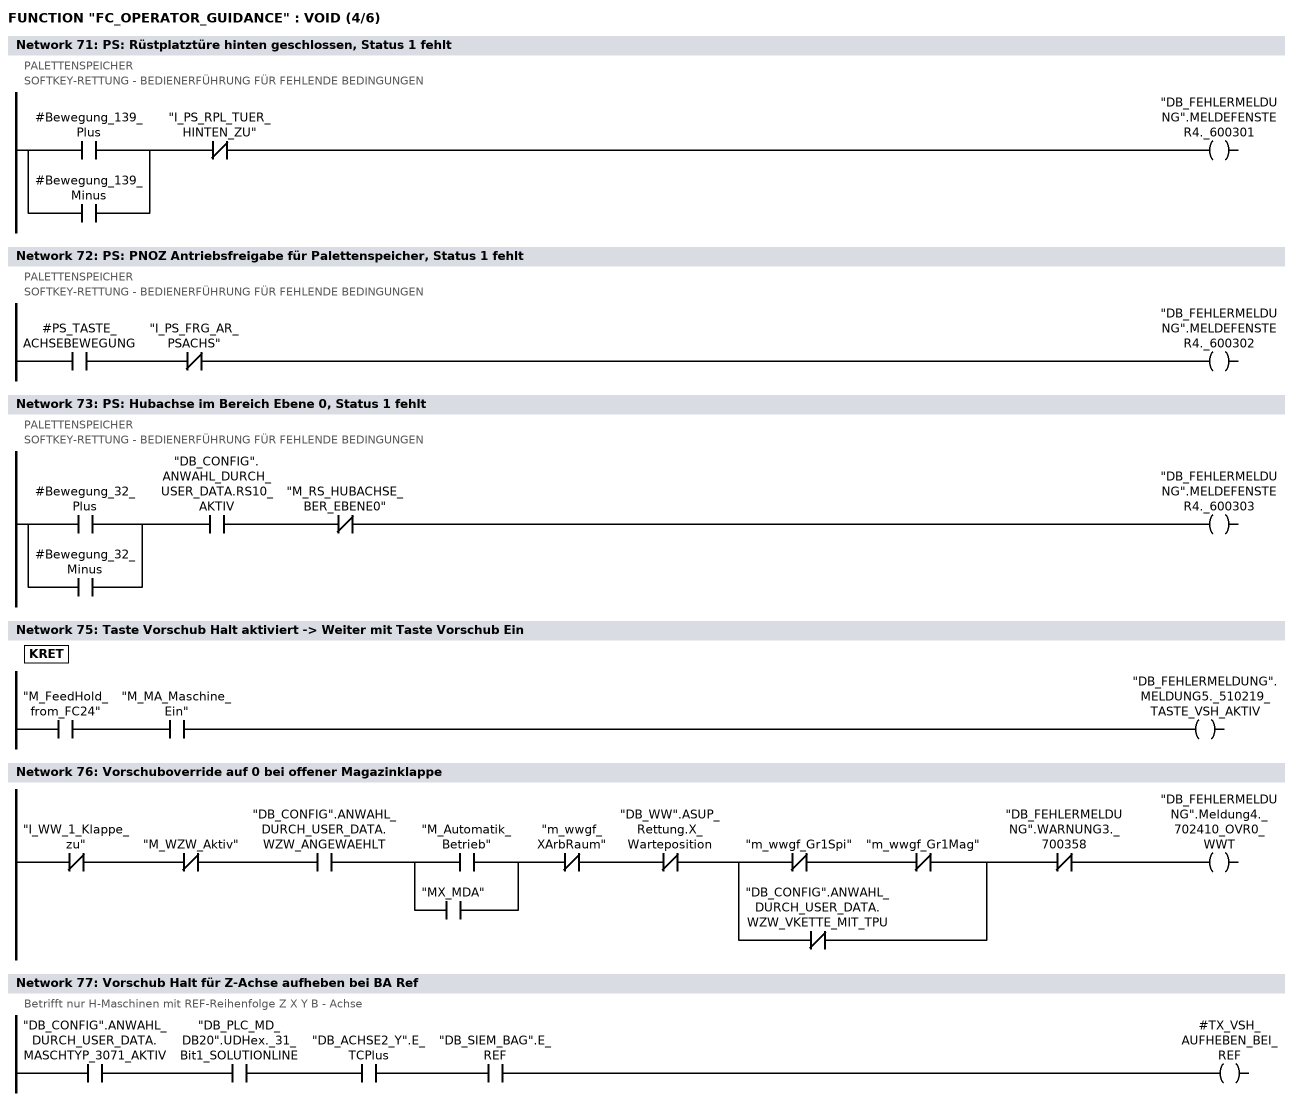
      U(    ;
      O     #Bewegung_139_Plus;
      O     #Bewegung_139_Minus;
      )     ;
      UN    "I_PS_RPL_TUER_HINTEN_ZU";
      =     "DB_FEHLERMELDUNG".MELDEFENSTER4._600301;
NETWORK
TITLE =PS: PNOZ Antriebsfreigabe für Palettenspeicher, Status 1 fehlt
//PALETTENSPEICHER
//SOFTKEY-RETTUNG - BEDIENERFÜHRUNG FÜR FEHLENDE BEDINGUNGEN
      U     #PS_TASTE_ACHSEBEWEGUNG;
      UN    "I_PS_FRG_AR_PSACHS";
      =     "DB_FEHLERMELDUNG".MELDEFENSTER4._600302;
NETWORK
TITLE =PS: Hubachse im Bereich Ebene 0, Status 1 fehlt
//PALETTENSPEICHER
//SOFTKEY-RETTUNG - BEDIENERFÜHRUNG FÜR FEHLENDE BEDINGUNGEN
      U(    ;
      O     #Bewegung_32_Plus;
      O     #Bewegung_32_Minus;
      )     ;
      U     "DB_CONFIG".ANWAHL_DURCH_USER_DATA.RS10_AKTIV;
      UN    "M_RS_HUBACHSE_BER_EBENE0";
      =     "DB_FEHLERMELDUNG".MELDEFENSTER4._600303;
NETWORK
TITLE =VORSCHUBSPERREN / VORSCHUB HALT

NETWORK
TITLE =Taste Vorschub Halt aktiviert -> Weiter mit Taste Vorschub Ein

KRET: U     "M_FeedHold_from_FC24";
      U     "M_MA_Maschine_Ein";
      =     "DB_FEHLERMELDUNG".MELDUNG5._510219_TASTE_VSH_AKTIV;
NETWORK
TITLE =Vorschuboverride auf 0 bei offener Magazinklappe

      UN    "I_WW_1_Klappe_zu";
      UN    "M_WZW_Aktiv";
      U     "DB_CONFIG".ANWAHL_DURCH_USER_DATA.WZW_ANGEWAEHLT;
      U(    ;
      O     "M_Automatik_Betrieb";
      O     "MX_MDA";
      )     ;
      UN    "m_wwgf_XArbRaum";
      UN    "DB_WW".ASUP_Rettung.X_Warteposition;
      U(    ;
      UN    "m_wwgf_Gr1Spi";
      UN    "m_wwgf_Gr1Mag";
      ON    "DB_CONFIG".ANWAHL_DURCH_USER_DATA.WZW_VKETTE_MIT_TPU;
      )     ;
      UN    "DB_FEHLERMELDUNG".WARNUNG3._700358;
      =     "DB_FEHLERMELDUNG".Meldung4._702410_OVR0_WWT;
NETWORK
TITLE =Vorschub Halt für Z-Achse aufheben bei BA Ref
//Betrifft nur H-Maschinen mit REF-Reihenfolge Z X Y B - Achse
      U     "DB_CONFIG".ANWAHL_DURCH_USER_DATA.MASCHTYP_3071_AKTIV;
      U     "DB_PLC_MD_DB20".UDHex._31_Bit1_SOLUTIONLINE;
      U     "DB_ACHSE2_Y".E_TCPlus;
      U     "DB_SIEM_BAG".E_REF;
      =     #TX_VSH_AUFHEBEN_BEI_REF;
NETWORK
TITLE =X-Achse im WZW Bereich -> Vorschub Halt an Y und Z Achse
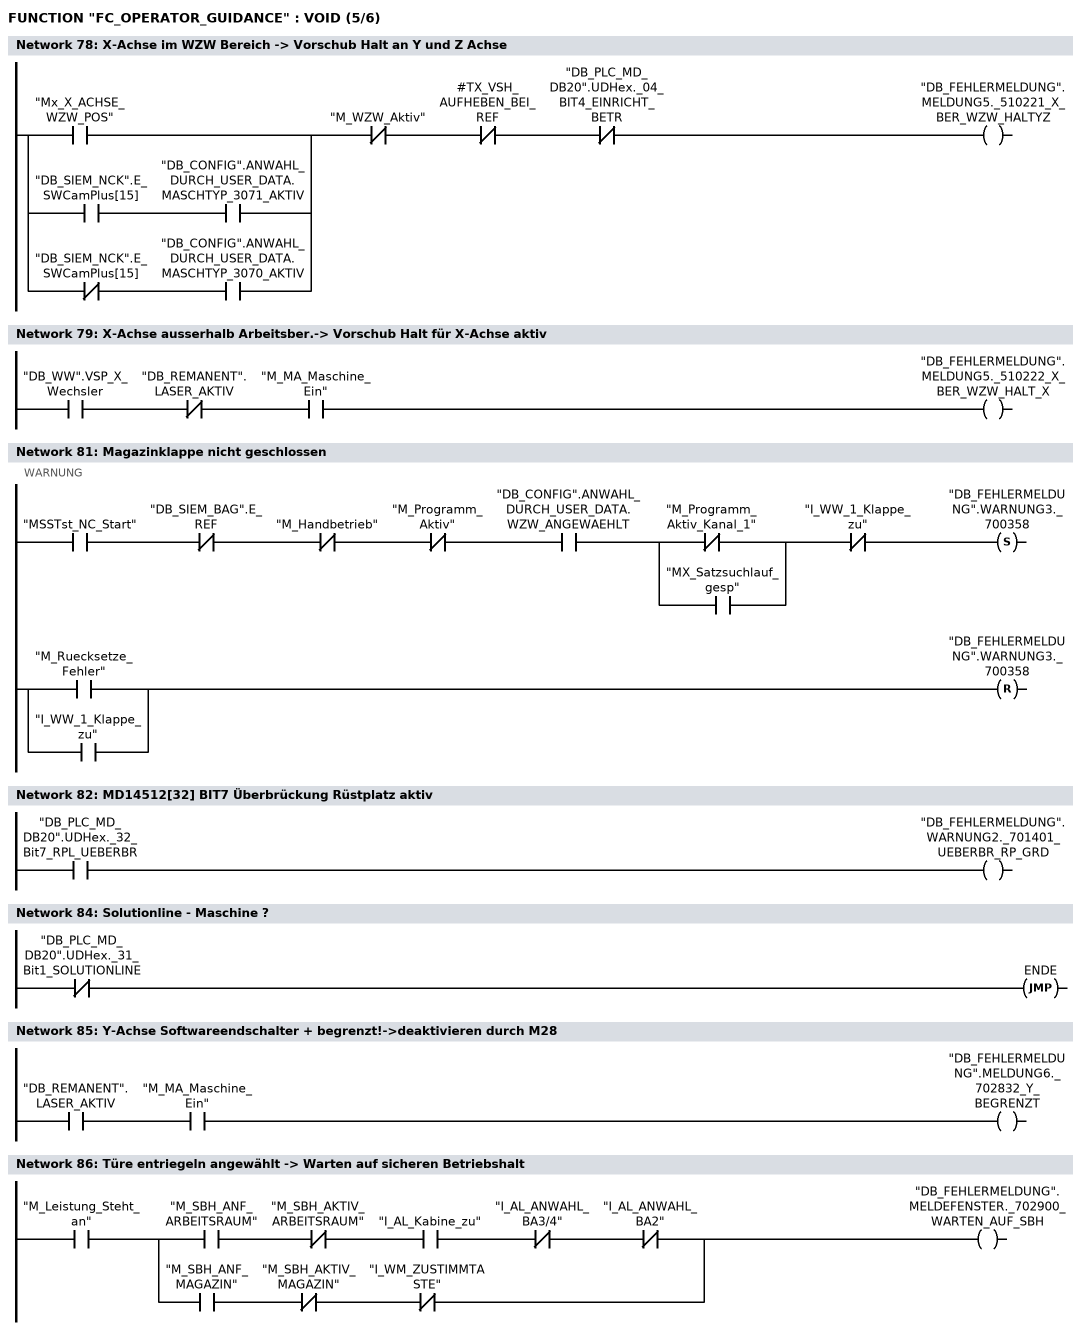

      U(    ;
      O     "Mx_X_ACHSE_WZW_POS";
      O     ;
      U     "DB_SIEM_NCK".E_SWCamPlus[15];
      U     "DB_CONFIG".ANWAHL_DURCH_USER_DATA.MASCHTYP_3071_AKTIV;
      O     ;
      UN    "DB_SIEM_NCK".E_SWCamPlus[15];
      U     "DB_CONFIG".ANWAHL_DURCH_USER_DATA.MASCHTYP_3070_AKTIV;
      )     ;
      UN    "M_WZW_Aktiv";
      UN    #TX_VSH_AUFHEBEN_BEI_REF;
      UN    "DB_PLC_MD_DB20".UDHex._04_BIT4_EINRICHT_BETR;
      =     "DB_FEHLERMELDUNG".MELDUNG5._510221_X_BER_WZW_HALTYZ;
NETWORK
TITLE =X-Achse ausserhalb Arbeitsber.-> Vorschub Halt für X-Achse aktiv

      U     "DB_WW".VSP_X_Wechsler;
      UN    "DB_REMANENT".LASER_AKTIV;
      U     "M_MA_Maschine_Ein";
      =     "DB_FEHLERMELDUNG".MELDUNG5._510222_X_BER_WZW_HALT_X;
NETWORK
TITLE =WARNUNGEN

NETWORK
TITLE =Magazinklappe nicht geschlossen
//WARNUNG
      U     "MSSTst_NC_Start";
      UN    "DB_SIEM_BAG".E_REF;
      UN    "M_Handbetrieb";
      UN    "M_Programm_Aktiv";
      U     "DB_CONFIG".ANWAHL_DURCH_USER_DATA.WZW_ANGEWAEHLT;
      U(    ;
      ON    "M_Programm_Aktiv_Kanal_1";
      O     "MX_Satzsuchlauf_gesp";
      )     ;
      UN    "I_WW_1_Klappe_zu";
      S     "DB_FEHLERMELDUNG".WARNUNG3._700358;
      U(    ;
      O     "M_Ruecksetze_Fehler";
      O     "I_WW_1_Klappe_zu";
      )     ;
      R     "DB_FEHLERMELDUNG".WARNUNG3._700358;
      NOP   0;
NETWORK
TITLE =MD14512[32] BIT7 Überbrückung Rüstplatz aktiv

      U     "DB_PLC_MD_DB20".UDHex._32_Bit7_RPL_UEBERBR;
      =     "DB_FEHLERMELDUNG".WARNUNG2._701401_UEBERBR_RP_GRD;

NETWORK
TITLE =SOLUTIONLINE ERWEITERTER DIAGNOSEBEREICH

NETWORK
TITLE =Solutionline - Maschine ?

      UN    "DB_PLC_MD_DB20".UDHex._31_Bit1_SOLUTIONLINE;
      SPB   ENDE;
NETWORK
TITLE =Y-Achse Softwareendschalter + begrenzt!->deaktivieren durch M28

      U     "DB_REMANENT".LASER_AKTIV;
      U     "M_MA_Maschine_Ein";
      =     "DB_FEHLERMELDUNG".MELDUNG6._702832_Y_BEGRENZT;
NETWORK
TITLE =Türe entriegeln angewählt -> Warten auf sicheren Betriebshalt

      U     "M_Leistung_Steht_an";
      U(    ;
      U     "M_SBH_ANF_ARBEITSRAUM";
      UN    "M_SBH_AKTIV_ARBEITSRAUM";
      U     "I_AL_Kabine_zu";
      UN    "I_AL_ANWAHL_BA3/4";
      UN    "I_AL_ANWAHL_BA2";
      O     ;
      U     "M_SBH_ANF_MAGAZIN";
      UN    "M_SBH_AKTIV_MAGAZIN";
      UN    "I_WM_ZUSTIMMTASTE";
      )     ;
      =     "DB_FEHLERMELDUNG".MELDEFENSTER._702900_WARTEN_AUF_SBH;
NETWORK
TITLE =Keine Rettungsfunktion aktiviert
//Info: DB101.DBX16.1 - 16.6  = Vertikale Rettungszeilen aktiviert
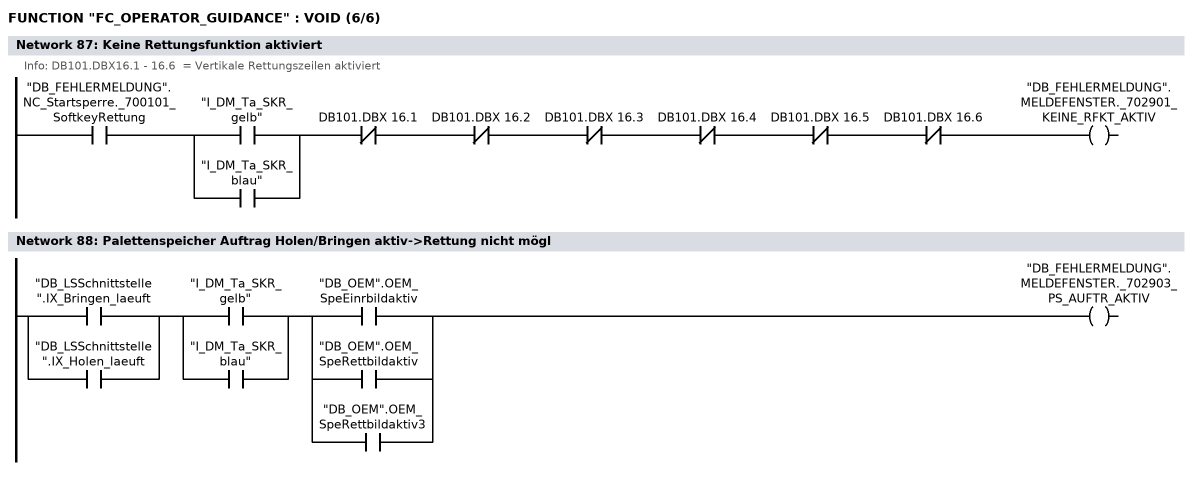
      U     "DB_FEHLERMELDUNG".NC_Startsperre._700101_SoftkeyRettung;
      U(    ;
      O     "I_DM_Ta_SKR_gelb";
      O     "I_DM_Ta_SKR_blau";
      )     ;
      UN    DB101.DBX   16.1;
      UN    DB101.DBX   16.2;
      UN    DB101.DBX   16.3;
      UN    DB101.DBX   16.4;
      UN    DB101.DBX   16.5;
      UN    DB101.DBX   16.6;
      =     "DB_FEHLERMELDUNG".MELDEFENSTER._702901_KEINE_RFKT_AKTIV;
NETWORK
TITLE =Palettenspeicher Auftrag Holen/Bringen aktiv->Rettung nicht mögl

      U(    ;
      O     "DB_LSSchnittstelle".IX_Bringen_laeuft;
      O     "DB_LSSchnittstelle".IX_Holen_laeuft;
      )     ;
      U(    ;
      O     "I_DM_Ta_SKR_gelb";
      O     "I_DM_Ta_SKR_blau";
      )     ;
      U(    ;
      O     "DB_OEM".OEM_SpeEinrbildaktiv;
      O     "DB_OEM".OEM_SpeRettbildaktiv;
      O     "DB_OEM".OEM_SpeRettbildaktiv3;
      )     ;
      =     "DB_FEHLERMELDUNG".MELDEFENSTER._702903_PS_AUFTR_AKTIV;
NETWORK
TITLE =Bausteinende

ENDE: NOP   0;

END_FUNCTION

